// TIA Portal V16 export
// export: Created 2021-11-12T13:33:01.9324613Z, ExportSetting WithDefaults, DisplayName Totally Integrated Automation Portal, DisplayVersion V16 Update 3, DisplayName TIA Portal Version Control Interface, DisplayVersion V16 Update 2, DisplayName TIA Portal Openness, DisplayVersion V16 Update 3, DisplayName SINAMICS Startdrive Advanced, DisplayVersion V16 Update 5, DisplayName SINAMICS Startdrive G130, G150, S120, S150, SINAMICS MV, S210, DisplayVersion V16 Update 5, DisplayName SINAMICS Startdrive G110M, G120, G120C, G120D, G120P, G115D, DisplayVersion V16 Update 5, DisplayName STEP 7 Professional, DisplayVersion V16 Update 3, DisplayName STEP 7 Safety, DisplayVersion V16, DisplayName WinCC UA Professional, DisplayVersion V16 Update 3
FUNCTION_BLOCK "Station430"   // FB54, LAD
{ S7_Optimized_Access := 'TRUE' }
VERSION : 0.1
// stored: AutoNumber true, IsIECCheckEnabled false, IsRetainMemResEnabled false, MemoryReserve 100, SetENOAutomatically false, UDAEnableTagReadback false
   VAR
      SF_GL01_MA01 : "STD_Drive1";
      SF_UC21_TA1 { S7_SetPoint := 'True'} : "STD_Siemens_G120_CU240E_2_PN";
      SF_Alarm1 { S7_SetPoint := 'True'} : "STD_DI_Mon";
      SF_Alarm2 { S7_SetPoint := 'True'} : "STD_DI_Mon";
      SF_OnOff { S7_SetPoint := 'True'} : "STD_OnOff";
      SF_TOF_BSN5 { S7_SetPoint := 'True'} : TOF_TIME;   // TOF timer to stop conv after BSN5 stopped
      SB1_PowerOk { S7_SetPoint := 'True'} : Bool;
   END_VAR
   VAR_TEMP
      TS_GL01MA01 : "UDT_DriveControl";
      TS_UC21TA01 : Struct
         ReqDir1 : Bool;   // Move in direction 1
         ReqDir2 : Bool;   // Move in direction 2
         AckErr : Bool;   // Acknowledge error
         SpeedSP : Real;   // Speed setpoint
      END_STRUCT;
      TB1_ConvBlock : Bool;   // Conveyor blocked
   END_VAR
BEGIN

REGION Network 1: ***************ClearTemporary***************
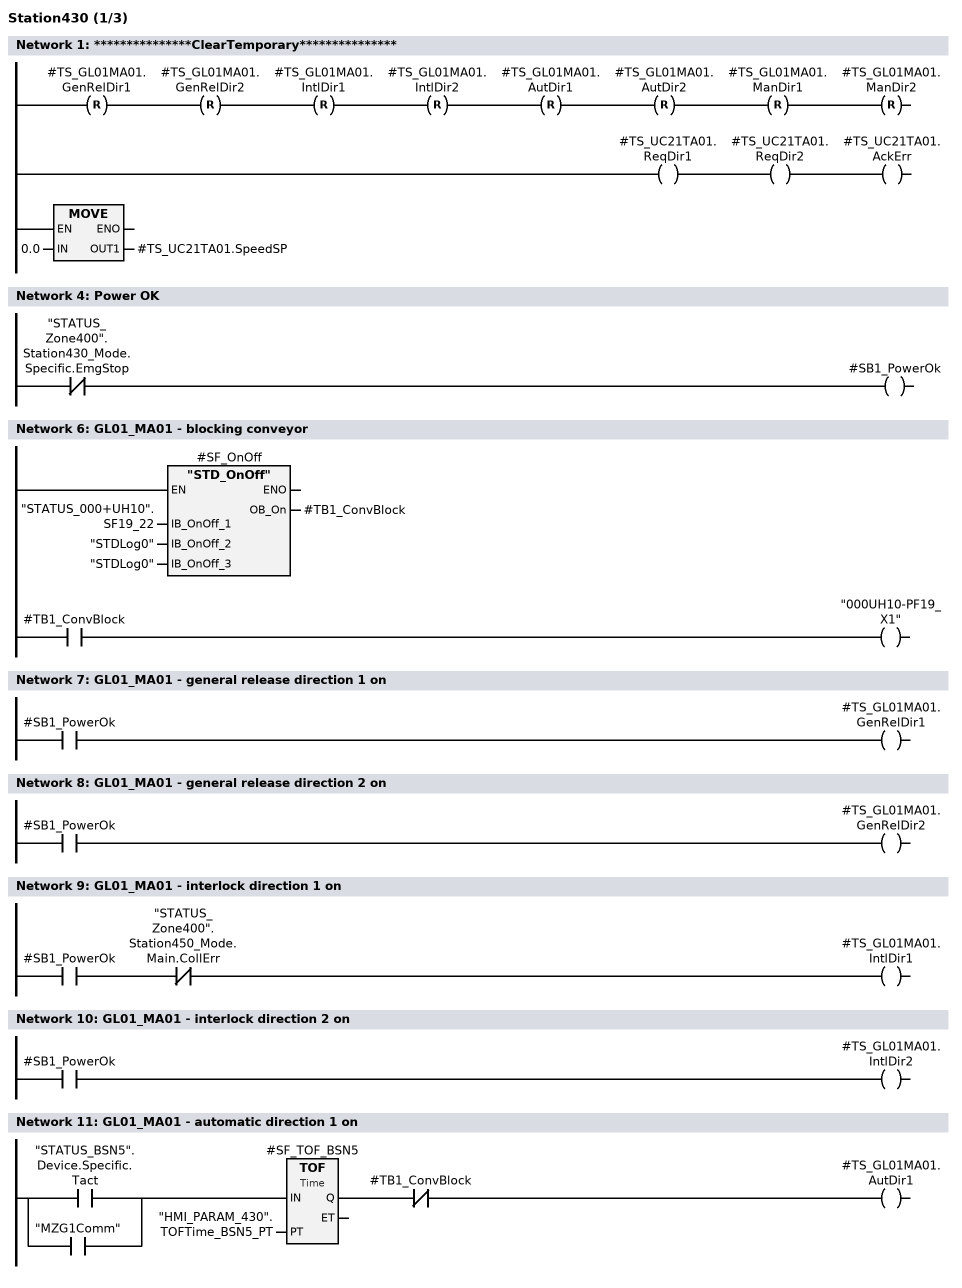
   RUNG wire#powerrail
      R_Coil( #TS_GL01MA01.GenRelDir1 )
      R_Coil( #TS_GL01MA01.GenRelDir2 )
      R_Coil( #TS_GL01MA01.IntlDir1 )
      R_Coil( #TS_GL01MA01.IntlDir2 )
      R_Coil( #TS_GL01MA01.AutDir1 )
      R_Coil( #TS_GL01MA01.AutDir2 )
      R_Coil( #TS_GL01MA01.ManDir1 )
      R_Coil( #TS_GL01MA01.ManDir2 )
   END_RUNG
   RUNG wire#powerrail
      Coil( #TS_UC21TA01.ReqDir1 )
      Coil( #TS_UC21TA01.ReqDir2 )
      Coil( #TS_UC21TA01.AckErr )
   END_RUNG
   RUNG wire#powerrail
      Move(in := 0.0, out1 => #TS_UC21TA01.SpeedSP)
   END_RUNG
   // the same network as SCL:
   #TS_GL01MA01.GenRelDir1 := FALSE;
   #TS_GL01MA01.GenRelDir2 := FALSE;
   #TS_GL01MA01.IntlDir1 := FALSE;
   #TS_GL01MA01.IntlDir2 := FALSE;
   #TS_GL01MA01.AutDir1 := FALSE;
   #TS_GL01MA01.AutDir2 := FALSE;
   #TS_GL01MA01.ManDir1 := FALSE;
   #TS_GL01MA01.ManDir2 := FALSE;
   #TS_UC21TA01.ReqDir1 := TRUE;
   #TS_UC21TA01.ReqDir2 := TRUE;
   #TS_UC21TA01.AckErr := TRUE;
   #TS_UC21TA01.SpeedSP := 0.0;
END_REGION

REGION Network 2: ***************SensorsAlarms***************
END_REGION

REGION Network 3: ***************ProcesAlarms***************
END_REGION

REGION Network 4: Power OK
   RUNG wire#powerrail
      I_Contact( "STATUS_Zone400".Station430_Mode.Specific.EmgStop )
      Coil( #SB1_PowerOk )
   END_RUNG
   // the same network as SCL:
   #SB1_PowerOk := NOT "STATUS_Zone400".Station430_Mode.Specific.EmgStop;
END_REGION

REGION Network 5: ***************GL01_MA01 Conveyor***************
END_REGION

REGION Network 6: GL01_MA01 - blocking conveyor
   RUNG wire#powerrail
      #SF_OnOff(IB_OnOff_1 := "STATUS_000+UH10".SF19_22, IB_OnOff_2 := "STDLog0", IB_OnOff_3 := "STDLog0", OB_On => #TB1_ConvBlock)
   END_RUNG
   RUNG wire#powerrail
      Contact( #TB1_ConvBlock )
      Coil( "000UH10-PF19_X1" )
   END_RUNG
   // the same network as SCL:
   #SF_OnOff(IB_OnOff_1 := "STATUS_000+UH10".SF19_22,   // "STD_OnOff"
             IB_OnOff_2 := "STDLog0",
             IB_OnOff_3 := "STDLog0",
             OB_On => #TB1_ConvBlock);
   "000UH10-PF19_X1" := #TB1_ConvBlock;
END_REGION

REGION Network 7: GL01_MA01 - general release direction 1 on
   RUNG wire#powerrail
      Contact( #SB1_PowerOk )
      Coil( #TS_GL01MA01.GenRelDir1 )
   END_RUNG
   // the same network as SCL:
   #TS_GL01MA01.GenRelDir1 := #SB1_PowerOk;
END_REGION

REGION Network 8: GL01_MA01 - general release direction 2 on
   RUNG wire#powerrail
      Contact( #SB1_PowerOk )
      Coil( #TS_GL01MA01.GenRelDir2 )
   END_RUNG
   // the same network as SCL:
   #TS_GL01MA01.GenRelDir2 := #SB1_PowerOk;
END_REGION

REGION Network 9: GL01_MA01 - interlock direction 1 on
   RUNG wire#powerrail
      Contact( #SB1_PowerOk )
      I_Contact( "STATUS_Zone400".Station450_Mode.Main.CollErr )
      Coil( #TS_GL01MA01.IntlDir1 )
   END_RUNG
   // the same network as SCL:
   #TS_GL01MA01.IntlDir1 := #SB1_PowerOk AND NOT "STATUS_Zone400".Station450_Mode.Main.CollErr;
END_REGION

REGION Network 10: GL01_MA01 - interlock direction 2 on
   RUNG wire#powerrail
      Contact( #SB1_PowerOk )
      Coil( #TS_GL01MA01.IntlDir2 )
   END_RUNG
   // the same network as SCL:
   #TS_GL01MA01.IntlDir2 := #SB1_PowerOk;
END_REGION

REGION Network 11: GL01_MA01 - automatic direction 1 on
   RUNG wire#powerrail
      Contact( "STATUS_BSN5".Device.Specific.Tact )
      wire#w1
      { S7_Templates := "time_type := Time" } #SF_TOF_BSN5.TOF(pt := "HMI_PARAM_430".TOFTime_BSN5_PT, et =>)
      I_Contact( #TB1_ConvBlock )
      Coil( #TS_GL01MA01.AutDir1 )
   END_RUNG
   RUNG wire#powerrail
      Contact( "MZG1Comm" )
   END_RUNG wire#w1
   // the same network as SCL:
   #SF_TOF_BSN5(IN := "STATUS_BSN5".Device.Specific.Tact OR "MZG1Comm", PT := "HMI_PARAM_430".TOFTime_BSN5_PT);   // TOF
   #TS_GL01MA01.AutDir1 := #SF_TOF_BSN5.Q AND NOT #TB1_ConvBlock;
END_REGION

REGION Network 12: GL01_MA01 - automatic direction 2 on
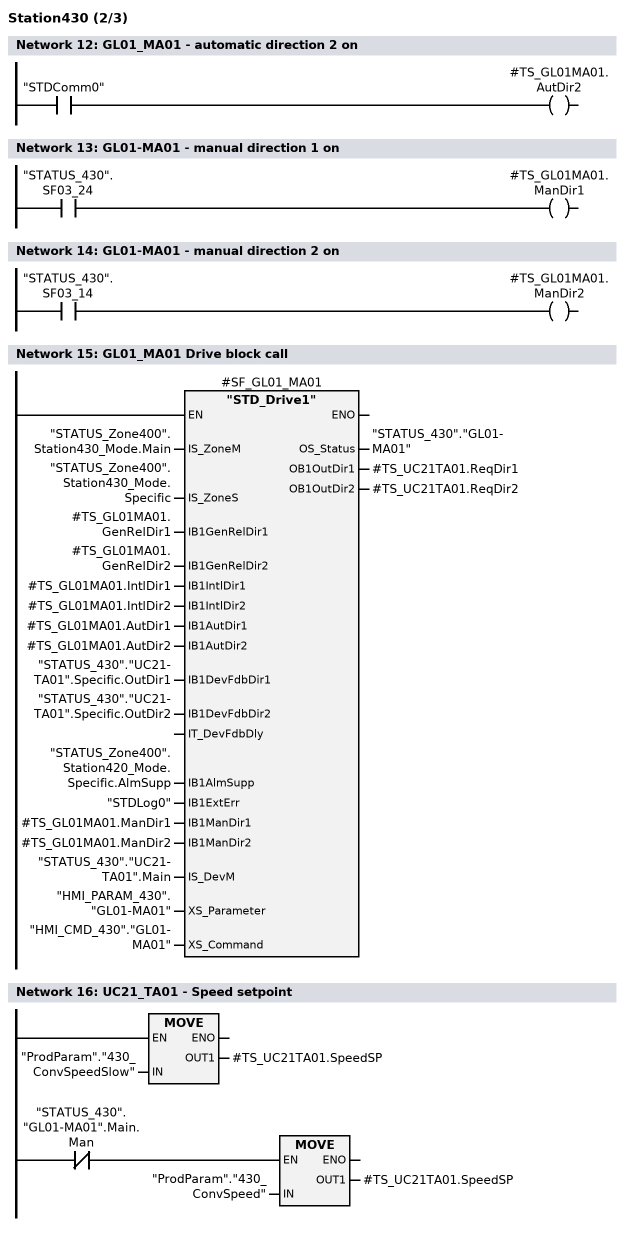
   RUNG wire#powerrail
      Contact( "STDComm0" )
      Coil( #TS_GL01MA01.AutDir2 )
   END_RUNG
   // the same network as SCL:
   #TS_GL01MA01.AutDir2 := "STDComm0";
END_REGION

REGION Network 13: GL01-MA01 - manual direction 1 on
   RUNG wire#powerrail
      Contact( "STATUS_430".SF03_24 )
      Coil( #TS_GL01MA01.ManDir1 )
   END_RUNG
   // the same network as SCL:
   #TS_GL01MA01.ManDir1 := "STATUS_430".SF03_24;
END_REGION

REGION Network 14: GL01-MA01 - manual direction 2 on
   RUNG wire#powerrail
      Contact( "STATUS_430".SF03_14 )
      Coil( #TS_GL01MA01.ManDir2 )
   END_RUNG
   // the same network as SCL:
   #TS_GL01MA01.ManDir2 := "STATUS_430".SF03_14;
END_REGION

REGION Network 15: GL01_MA01 Drive block call
   RUNG wire#powerrail
      #SF_GL01_MA01(IS_ZoneM := "STATUS_Zone400".Station430_Mode.Main, IS_ZoneS := "STATUS_Zone400".Station430_Mode.Specific, IB1GenRelDir1 := #TS_GL01MA01.GenRelDir1, IB1GenRelDir2 := #TS_GL01MA01.GenRelDir2, IB1IntlDir1 := #TS_GL01MA01.IntlDir1, IB1IntlDir2 := #TS_GL01MA01.IntlDir2, IB1AutDir1 := #TS_GL01MA01.AutDir1, IB1AutDir2 := #TS_GL01MA01.AutDir2, IB1DevFdbDir1 := "STATUS_430"."UC21-TA01".Specific.OutDir1, IB1DevFdbDir2 := "STATUS_430"."UC21-TA01".Specific.OutDir2, IT_DevFdbDly :=, IB1AlmSupp := "STATUS_Zone400".Station420_Mode.Specific.AlmSupp, IB1ExtErr := "STDLog0", IB1ManDir1 := #TS_GL01MA01.ManDir1, IB1ManDir2 := #TS_GL01MA01.ManDir2, IS_DevM := "STATUS_430"."UC21-TA01".Main, XS_Parameter := "HMI_PARAM_430"."GL01-MA01", XS_Command := "HMI_CMD_430"."GL01-MA01", OS_Status => "STATUS_430"."GL01-MA01", OB1OutDir1 => #TS_UC21TA01.ReqDir1, OB1OutDir2 => #TS_UC21TA01.ReqDir2)
   END_RUNG
   // the same network as SCL:
   #SF_GL01_MA01(IS_ZoneM := "STATUS_Zone400".Station430_Mode.Main,   // "STD_Drive1"
                 IS_ZoneS := "STATUS_Zone400".Station430_Mode.Specific,
                 IB1GenRelDir1 := #TS_GL01MA01.GenRelDir1,
                 IB1GenRelDir2 := #TS_GL01MA01.GenRelDir2,
                 IB1IntlDir1 := #TS_GL01MA01.IntlDir1,
                 IB1IntlDir2 := #TS_GL01MA01.IntlDir2,
                 IB1AutDir1 := #TS_GL01MA01.AutDir1,
                 IB1AutDir2 := #TS_GL01MA01.AutDir2,
                 IB1DevFdbDir1 := "STATUS_430"."UC21-TA01".Specific.OutDir1,
                 IB1DevFdbDir2 := "STATUS_430"."UC21-TA01".Specific.OutDir2,
                 IB1AlmSupp := "STATUS_Zone400".Station420_Mode.Specific.AlmSupp,
                 IB1ExtErr := "STDLog0",
                 IB1ManDir1 := #TS_GL01MA01.ManDir1,
                 IB1ManDir2 := #TS_GL01MA01.ManDir2,
                 IS_DevM := "STATUS_430"."UC21-TA01".Main,
                 XS_Parameter := "HMI_PARAM_430"."GL01-MA01",
                 XS_Command := "HMI_CMD_430"."GL01-MA01",
                 OS_Status => "STATUS_430"."GL01-MA01",
                 OB1OutDir1 => #TS_UC21TA01.ReqDir1,
                 OB1OutDir2 => #TS_UC21TA01.ReqDir2);
END_REGION

REGION Network 16: UC21_TA01 - Speed setpoint
   RUNG wire#powerrail
      Move(in := "ProdParam"."430_ConvSpeedSlow", out1 => #TS_UC21TA01.SpeedSP)
   END_RUNG
   RUNG wire#powerrail
      I_Contact( "STATUS_430"."GL01-MA01".Main.Man )
      Move(in := "ProdParam"."430_ConvSpeed", out1 => #TS_UC21TA01.SpeedSP)
   END_RUNG
   // the same network as SCL:
   #TS_UC21TA01.SpeedSP := "ProdParam"."430_ConvSpeedSlow";
   IF NOT "STATUS_430"."GL01-MA01".Main.Man THEN #TS_UC21TA01.SpeedSP := "ProdParam"."430_ConvSpeed"; END_IF;
END_REGION

REGION Network 17: UC21_TA01 - Frequency convertor block call
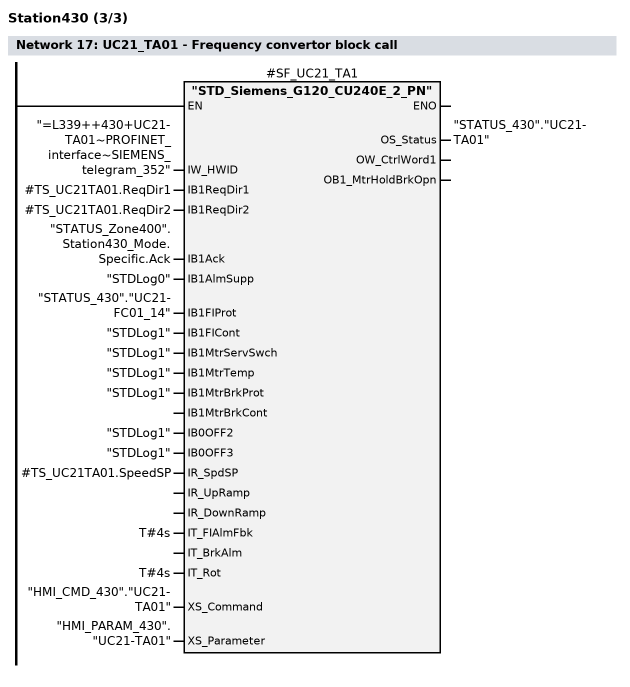
   RUNG wire#powerrail
      #SF_UC21_TA1(IW_HWID := "=L339++430+UC21-TA01~PROFINET_interface~SIEMENS_telegram_352", IB1ReqDir1 := #TS_UC21TA01.ReqDir1, IB1ReqDir2 := #TS_UC21TA01.ReqDir2, IB1Ack := "STATUS_Zone400".Station430_Mode.Specific.Ack, IB1AlmSupp := "STDLog0", IB1FIProt := "STATUS_430"."UC21-FC01_14", IB1FICont := "STDLog1", IB1MtrServSwch := "STDLog1", IB1MtrTemp := "STDLog1", IB1MtrBrkProt := "STDLog1", IB1MtrBrkCont :=, IB0OFF2 := "STDLog1", IB0OFF3 := "STDLog1", IR_SpdSP := #TS_UC21TA01.SpeedSP, IR_UpRamp :=, IR_DownRamp :=, IT_FIAlmFbk := T#4s, IT_BrkAlm :=, IT_Rot := T#4s, XS_Command := "HMI_CMD_430"."UC21-TA01", XS_Parameter := "HMI_PARAM_430"."UC21-TA01", OS_Status => "STATUS_430"."UC21-TA01", OW_CtrlWord1 =>, OB1_MtrHoldBrkOpn =>)
   END_RUNG
   // the same network as SCL:
   #SF_UC21_TA1(IW_HWID := "=L339++430+UC21-TA01~PROFINET_interface~SIEMENS_telegram_352",   // "STD_Siemens_G120_CU240E_2_PN"
                IB1ReqDir1 := #TS_UC21TA01.ReqDir1,
                IB1ReqDir2 := #TS_UC21TA01.ReqDir2,
                IB1Ack := "STATUS_Zone400".Station430_Mode.Specific.Ack,
                IB1AlmSupp := "STDLog0",
                IB1FIProt := "STATUS_430"."UC21-FC01_14",
                IB1FICont := "STDLog1",
                IB1MtrServSwch := "STDLog1",
                IB1MtrTemp := "STDLog1",
                IB1MtrBrkProt := "STDLog1",
                IB0OFF2 := "STDLog1",
                IB0OFF3 := "STDLog1",
                IR_SpdSP := #TS_UC21TA01.SpeedSP,
                IT_FIAlmFbk := T#4s,
                IT_Rot := T#4s,
                XS_Command := "HMI_CMD_430"."UC21-TA01",
                XS_Parameter := "HMI_PARAM_430"."UC21-TA01",
                OS_Status => "STATUS_430"."UC21-TA01");
END_REGION
END_FUNCTION_BLOCK
